PROGRAM MAIN_OLD 
VAR 
	fbMotorJog			:	FB_MotorJog;
	fbCamera			:	FB_Camera;
	fbMagStirrer		:	FB_MagStirrer;
// 	fbQRcode			:	FB_Camera;
// 	fbTest 				: FB_Test;
	fbEL6001			: FB_SerialCom;
	
	plcIN0 AT%I* : ARRAY [0..7] OF UINT;	//inputs w.r.t. PLC
	plcIN1 AT%I* : ARRAY [0..7] OF UINT;	
	plcIN2 AT%I* : ARRAY [0..7] OF UINT;
	plcIN3 AT%I* : ARRAY [0..7] OF UINT;

	plcOUT1 AT%Q* : ARRAY [0..7] OF UINT;	//outputs w.r.t. PLC
	plcOUT2 AT%Q* : ARRAY [0..7] OF UINT;
	plcOUT3 AT%Q* : ARRAY [0..7] OF UINT;	
	plcOUT0 AT%Q* : ARRAY [0..7] OF UINT;	
	bIndex				:	USINT	:=2;
	fSuccess: BOOL;
	
	bTrigHome : BOOL;
	bTrigGrip : BOOL;
	
	bFunctionality : INT:=0;
	
	bFlag: BOOL;
	trigHome : R_TRIG;

END_VAR

// fbTest();
fbCamera.TriggerCamera();
// fbMotorJog.CapContainer();
// fSuccess := fbSoftwareTrigger.DetectQRCode();	
	
	plcIN0[4].0;			// DO145
	plcIN1[0].0;		// DO209	
	plcOUT1[0].0;		// DI209 
	plcOUT1[0].1;		// DI210
	plcOUT1[0].2;		// DI211
	
	CASE bFunctionality OF
		0: 
			plcOUT1[0].0:=FALSE;
			plcOUT1[0].1:=FALSE;
			IF bFlag THEN
				bFunctionality:=10;
			END_IF
	
		10:
			plcOUT1[0].0:=TRUE;			// Trigger Move to Home
			trigHome(CLK := plcIN1[0].8);
			IF trigHome.Q THEN 
				plcOUT1[0].0:=FALSE;
				bFunctionality:=20;
			END_IF
			
		20:
			plcOUT1[0].1:=TRUE;			// Trigger Grip fingers
			IF plcIN1[0].8=TRUE THEN
				plcOUT1[0].1:=FALSE;	// 
			END_IF
				
	END_CASE

// hr := F_VN_ReadQRCodeExp(ipImageIn, ipDecodedData, ipContours, nCodeNumber,
// 		 eSearchStrategy, hr);
// 		 
// hr := F_VN_DrawContours(ipCodeContourList, 0, ipImageRes, aColorRed, 3, hr);

ACTION GripFingersAB:
(*-- program to trigger gripping of fingers on Schunk Deposit Station A and B --*)

(*Initialize Inputs to OFF for every PLC cycle*)
plcOUT0[4].0:=FALSE;	// DI145 
plcOUT0[4].1:=FALSE;	// DI146


// IF bTrigGrip THEN				// If DO209=ON state trigger state 'grip fingers AB' is true
	plcOUT1[0].1:=TRUE;					// Then DI210=ON && Triggers the program in the TP for gripper change
// 		
// 	IF plcIN1[0].8:=TRUE THEN			// DO217=ON && get input whether Gripper change TP program is Successfully completed
// 		plcOUT1[0].1:=FALSE;			// Turn off TPprogram trigger when successfully completed
// 	ELSE
// 		plcOUT0[4].1:=TRUE;				// Error state DI146 is turned to ON
// 	END_IF
// 	bTrigGrip := FALSE;
// END_IF
END_ACTION

ACTION MoveToHome:
(*-- program to move Robot to Home Pose --*)

(*Initialize Inputs to OFF for every PLC cycle*)
plcOUT0[4].0:=FALSE;	// DI145 
plcOUT0[4].1:=FALSE;	// DI146

// IF bTrigHome THEN				// If DO209=ON state trigger state 'move to home' is true
	plcOUT1[0].0:=TRUE;					// Then DI209=ON && Triggers the program in the TP for moving to home pose
// 		
// 	IF plcIN1[0].8:=TRUE THEN			// DO217=ON && get input whether Gripper change TP program is Successfully completed
// 		plcOUT1[0].1:=FALSE;			// Turn off TPprogram trigger when successfully completed
// 	ELSE
// 		plcOUT0[4].1:=TRUE;				// Error state DI146 is turned to ON
// 	END_IF
// 	bTrigHome := FALSE;
// END_IF
END_ACTION

END_PROGRAM

(* stored: Version 1.1.0.1
   POU MAIN_OLD: Id {5ffd7926-5d16-4ef4-80ac-73e67cfe458d}, SpecialFunc None
   Action GripFingersAB: Id {54710d87-64ea-43a9-bfa1-ed109fbc33f7}
   Action MoveToHome: Id {85e6d515-854e-4ccf-aadd-b310af254146} *)
